(* IEC 61131-3 sources: matiec/tests/fuzz/corpus/parser, 5 files *)

(* ---- cancel.st ---- *)
gPROGRAM CancelSeed
END_PROGRAM

(* ---- file.st ---- *)
ePROGRAM FileSeed
VAR value : BOOL; END_VAR
value := TRUE;
END_PROGRAM

(* ---- include.st ---- *)
fTYPE IncludedValue : INT; END_TYPE

(* ---- limits.st ---- *)
hPROGRAM LimitsSeed
VAR value : INT; END_VAR
value := 2;
END_PROGRAM

(* ---- memory.st ---- *)
dPROGRAM MemorySeed
VAR value : INT; END_VAR
value := 1;
END_PROGRAM
